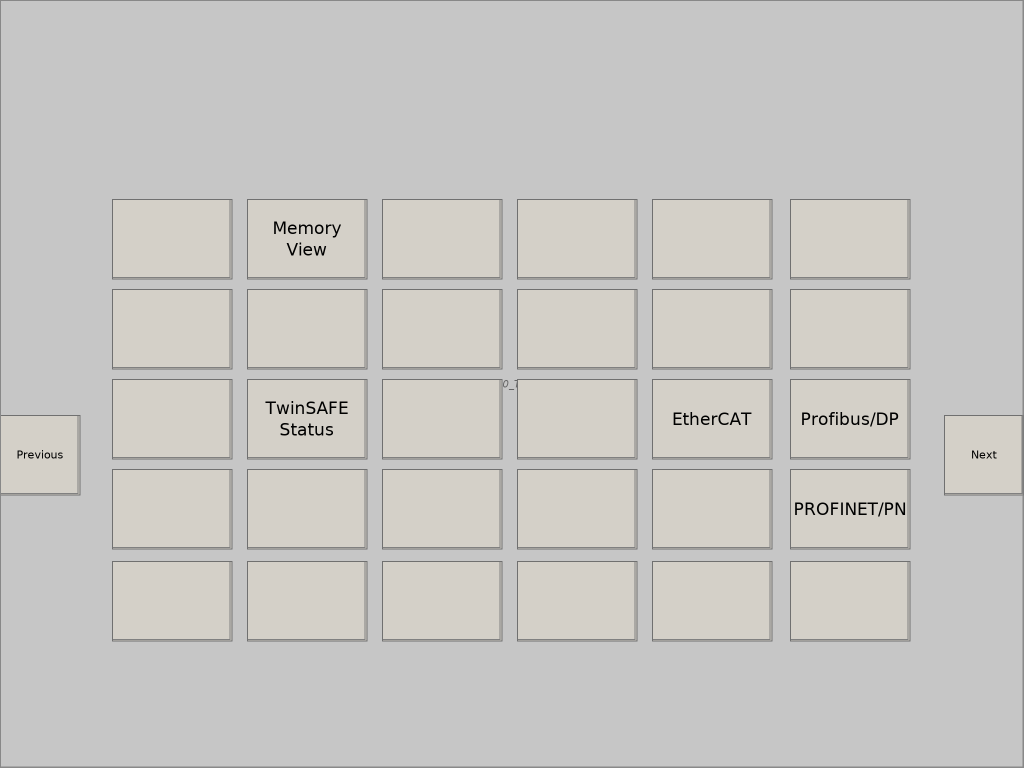
VISUALIZATION Men_031_MenuScreen_2  // 1024x768
    Frame (0,0 1024x768)
        shows Tmp_000_Template(header := gHMIData.hmiHeader)
    Button (112,199 120x80), text list: ''
    Button (247,199 120x80), "Memory View", text list: ''
        OnMouseClick: change screen: Dia_800_DataDisplay
    Button (382,199 120x80), text list: ''
    Button (517,199 120x80), text list: ''
    Button (652,199 120x80), text list: ''
    Button (790,199 120x80), text list: ''
    Button (112,289 120x80), text list: ''
    Button (247,289 120x80), text list: ''
    Button (382,289 120x80), text list: ''
    Button (517,289 120x80), text list: ''
    Button (652,289 120x80), text list: ''
    Button (790,289 120x80), text list: ''
    Button (112,379 120x80), text list: ''
    Button (247,379 120x80), "TwinSAFE Status", text list: ''
        OnMouseClick: change screen: Saf_700_SafetyStatus
    Button (382,379 120x80), text list: ''
    Button (517,379 120x80), text list: ''
    Button (652,379 120x80), "EtherCAT", text list: ''
        OnMouseClick: change screen: Dia_801_EtherCAT
    Button (790,379 120x80), "Profibus/DP", text list: ''
        OnMouseClick: change screen: Dia_802_Profibus
    Button (112,469 120x80), text list: ''
    Button (247,469 120x80), text list: ''
    Button (382,469 120x80), text list: ''
    Button (517,469 120x80), text list: ''
    Button (652,469 120x80), text list: ''
    Button (790,469 120x80), "PROFINET/PN", text list: ''
        OnMouseClick: change screen: Dia_803_ProfiNet
    Button (112,561 120x80), text list: ''
    Button (247,561 120x80), text list: ''
    Button (382,561 120x80), text list: ''
    Button (517,561 120x80), text list: ''
    Button (652,561 120x80), text list: ''
    Button (790,561 120x80), text list: ''
    Group (0,415 1024x80)
        Button (0,0 80x80), "Previous"
            OnMouseClick: change screen: Men_030_MenuScreen
        Button (944,0 80x80), "Next"
            OnMouseClick: change screen: Men_032_MenuScreen_3
END_VISUALIZATION

(* stored: Version 1.1.0.1, ProductVersion 3.1.4024.11
   Visu Men_031_MenuScreen_2: Id {bb8a863c-ae30-4809-9425-2739f868bb94} *)
